Omron CX-Programmer project NewProject (CX-Programmer 9.73)

# PLC NewPLC1: CP1E E20

## Global symbols (name address type ; comment)
100.05 BOOL  ; Robot Arm 2
100.04 BOOL  ; Robot Arm 1
100.03 BOOL  ; Sanitizing Spray
0.00 BOOL  ; Start / Reset
0.01 BOOL  ; Sensor 1
0.02 BOOL  ; Sensor 2
0.03 BOOL  ; Stop
0.04 BOOL  ; OFF
100.00 BOOL  ; Conveyor1
100.01 BOOL  ; Conveyor 1
100.02 BOOL  ; Conveyor 2
C000 BOOL  ; Counter1
C001 BOOL  ; Counter 1
C002 BOOL  ; Counter 2
C003 BOOL  ; Counter3
T001 BOOL  ; Timer 1
T002 BOOL  ; Timer 2
W0.00 BOOL  ; Activation Relay
W0.01 BOOL  ; Relay 1
W0.02 BOOL  ; Relay 2
W0.03 BOOL  ; OffRobot1
W0.04 BOOL  ; OffRobot2

## Program NewProgram1 (cyclic task 0)

### Section Section1

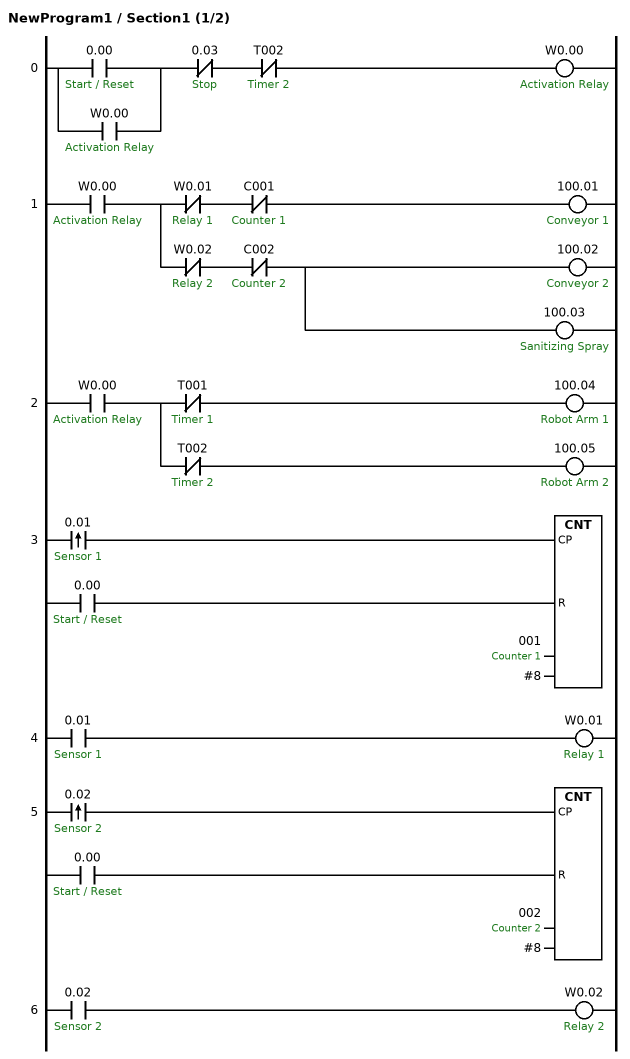
; rung 0
LD 0.00  ; Start / Reset
OR W0.00  ; Activation Relay
ANDNOT 0.03  ; Stop
ANDNOT T002  ; Timer 2
OUT W0.00  ; Activation Relay
; rung 1
LD W0.00  ; Activation Relay
OUT TR0
ANDNOT W0.01  ; Relay 1
ANDNOT C001  ; Counter 1
OUT 100.01  ; Conveyor 1
LD TR0
ANDNOT W0.02  ; Relay 2
ANDNOT C002  ; Counter 2
OUT 100.02  ; Conveyor 2
OUT 100.03  ; Sanitizing Spray
; rung 2
LD W0.00  ; Activation Relay
OUT TR0
ANDNOT T001  ; Timer 1
OUT 100.04  ; Robot Arm 1
LD TR0
ANDNOT T002  ; Timer 2
OUT 100.05  ; Robot Arm 2
; rung 3
@LD 0.01  ; Sensor 1
LD 0.00  ; Start / Reset
CNT 001 #8  ; Counter 1
; rung 4
LD 0.01  ; Sensor 1
OUT W0.01  ; Relay 1
; rung 5
@LD 0.02  ; Sensor 2
LD 0.00  ; Start / Reset
CNT 002 #8  ; Counter 2
; rung 6
LD 0.02  ; Sensor 2
OUT W0.02  ; Relay 2

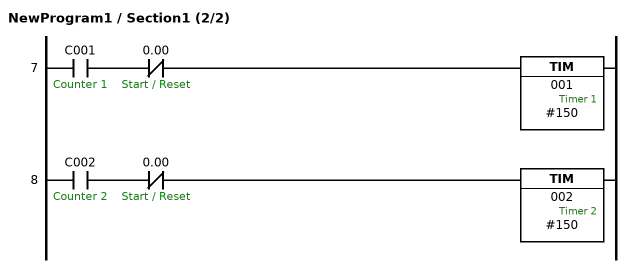
; rung 7
LD C001  ; Counter 1
ANDNOT 0.00  ; Start / Reset
TIM 001 #150  ; Timer 1
; rung 8
LD C002  ; Counter 2
ANDNOT 0.00  ; Start / Reset
TIM 002 #150  ; Timer 2

### Section END
; rung 0
END(001)